TYPE ST_EL9110 :
STRUCT
	PowerOK							AT %I*	:BOOL;
	State							AT %I*	:UINT;
END_STRUCT
END_TYPE

(* stored: Version 1.1.0.1
   DUT ST_EL9110: Id {50d355ae-b950-418b-acaa-fcc97ef0cd75} *)
